// TIA Portal V17 export
// export: Created 2021-12-03T08:12:55.7140446Z, ExportSetting WithDefaults, DisplayName Totally Integrated Automation Portal, DisplayVersion V17, DisplayName TIA Portal Openness, DisplayVersion V17, DisplayName TIA Portal Version Control Interface, DisplayVersion V17, DisplayName STEP 7 Professional, DisplayVersion V17, DisplayName STEP 7 Safety, DisplayVersion V17, DisplayName WinCC Advanced, DisplayVersion V17
FUNCTION_BLOCK "FB_DetLineSts"   // FB22, FBD
VERSION : 0.1
// stored: AutoNumber false, IsIECCheckEnabled false, UDAEnableTagReadback false
   VAR_INPUT
      ID { ExternalVisible := 'False'} : Int;
      LADDR { ExternalVisible := 'False'} : Word;
      I_FltAck { ExternalVisible := 'False'} : Bool;
   END_VAR
   VAR_OUTPUT
      O_ConOk { ExternalVisible := 'False'; ExternalWritable := 'False'} : Bool;   // 1=Detector Line Connected
      O_SyncStrt { ExternalVisible := 'False'; ExternalWritable := 'False'} : Bool;   // 1=Synchronizator Started
      O_ScanAct { ExternalVisible := 'False'; ExternalWritable := 'False'} : Bool;   // 1=Scanning active
      O_RdyForScan { ExternalVisible := 'False'; ExternalWritable := 'False'} : Bool;   // 1=Ready for scanning
      O_ErrRdyAck { ExternalVisible := 'False'; ExternalWritable := 'False'} : Bool;   // 1=Error ready ack
      O_State { ExternalVisible := 'False'; ExternalWritable := 'False'} : Int;   // State: 0=Error, 1=Service mode, 2=OK
      O_ErgMd { ExternalVisible := 'False'; ExternalWritable := 'False'} : Int;   // Energy Mode: 0=Reserved, 1=Low, 2=High, 3=Dual energy)
      O_TrigRate { ExternalVisible := 'False'; ExternalWritable := 'False'} : Int;   // Trigger Rate (Range 50-1000, Step 1)
   END_VAR
   VAR DB_SPECIFIC
      DetLine_Sts { ExternalVisible := 'False'; ExternalWritable := 'False'} : Struct
         MsgId { ExternalVisible := 'False'; ExternalWritable := 'False'} : DWord;   // Message Id
         MsgLen { ExternalVisible := 'False'; ExternalWritable := 'False'} : DWord;   // Message Length
         Sts { ExternalVisible := 'False'; ExternalWritable := 'False'} : DWord;   // Status
         State { ExternalVisible := 'False'; ExternalWritable := 'False'} : DWord;   // State: 0=Error, 1=Service mode, 2=OK
         ErgMode { ExternalVisible := 'False'; ExternalWritable := 'False'} : DWord;   // Energy Mode: 0=Reserved, 1=Low, 2=High, 3=Dual energy)
         TrigRate { ExternalVisible := 'False'; ExternalWritable := 'False'} : DWord;   // Trigger Rate (Range 50-1000, Step 1)
      END_STRUCT;
      TCP_Sts { ExternalVisible := 'False'} : Struct
         Done { ExternalVisible := 'False'} : Bool;
         Error { ExternalVisible := 'False'} : Bool;
         Status { ExternalVisible := 'False'} : Word;
         Len { ExternalVisible := 'False'} : Int;
         ErrCd { ExternalVisible := 'False'} : Word;
      END_STRUCT;
      AxPtrig { ExternalVisible := 'False'} : Struct
         Done { ExternalVisible := 'False'} : Bool;
      END_STRUCT;
      S_AckRq { ExternalVisible := 'False'} : Bool;
      S_Con_Nok { ExternalVisible := 'False'} : Bool;
   END_VAR
   VAR_TEMP   // added for the SCL form of the ladder/FBD networks
      _w1 : Bool;
   END_VAR
BEGIN

REGION Network 1: Блок чтения данных с Detector Module
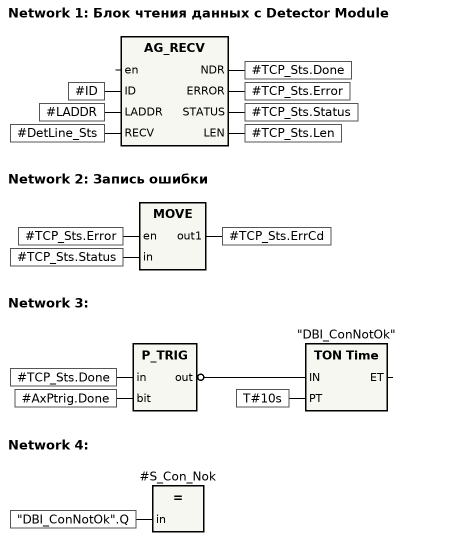
   AG_RECV(ID := #ID,
           LADDR := #LADDR,
           RECV := #DetLine_Sts,
           NDR => #TCP_Sts.Done,
           ERROR => #TCP_Sts.Error,
           STATUS => #TCP_Sts.Status,
           LEN => #TCP_Sts.Len);
END_REGION

REGION Network 2: Запись ошибки
   IF #TCP_Sts.Error THEN #TCP_Sts.ErrCd := #TCP_Sts.Status; END_IF;
END_REGION

REGION Network 3
   #_w1 := #TCP_Sts.Done AND NOT #AxPtrig.Done;   // rising edge
   #AxPtrig.Done := #TCP_Sts.Done;
   "DBI_ConNotOk".TON(IN := NOT #_w1, PT := T#10s);
END_REGION

REGION Network 4
   #S_Con_Nok := "DBI_ConNotOk".Q;
END_REGION

NETWORK
TITLE = Копирование статусов
      L     #DetLine_Sts.Sts;
      T     "DetLineSts_Sts";

      AN    #S_Con_Nok;
      =     #O_ConOk;

      A     "DetLineSts_SyncStrt";
      =     #O_SyncStrt;

      A     "DetLineSts_ScanAct";
      =     #O_ScanAct;

      A     "DetLineSts_RdyForScan";
      =     #O_RdyForScan;

      L     #DetLine_Sts.State;
      T     #O_State;

      L     #DetLine_Sts.ErgMode;
      T     #O_ErgMd;

      L     #DetLine_Sts.TrigRate;
      T     #O_TrigRate;
END_FUNCTION_BLOCK
